TYPE InfoDataAdsAddrStateBase_1916E49F :
STRUCT
END_STRUCT
END_TYPE

(* stored: Version 1.2.0.0, ProductVersion 3.1.4024.9
   DUT InfoDataAdsAddrStateBase_1916E49F: Id {5bcf7446-4898-49dd-9517-c33f7a681d74} *)
